Fanuc KAREL source: GET_QUEUE.kl

PROGRAM T
%NOLOCKGROUP
VAR
 v0 : QUEUE_TYPE
 v1 : ARRAY[10] OF INTEGER
 v2 : INTEGER
 v3 : INTEGER
 v4 : INTEGER
BEGIN
 GET_QUEUE(v0, v1, v2, v3, v4)
END T
